PROGRAM MAIN
VAR
END_VAR

END_PROGRAM

(* stored: Version 1.1.0.1
   POU MAIN: Id {d694e92c-10ba-48b4-b5f0-9adc81d2091c} *)
